PROGRAM PMPS_Arbiter
VAR
	
	fbPhotonEnergyWatcher	:	FB_PhotonEnergyWatcher;
	
	fbMPSInterface	:	FB_BeamClassOutputs;
    
    fbCuInterface	:	FB_CTLS_Outputs;
	
	(* Subsystem requests use this FB and a pragma link to pass their requests to the arbiter.
	The fb is called on each cycle and updates the arbiter with the current BP set requested 
	from the subsystem PLC.*)
	//<TODO> make this so it does input and output to the IF
	{attribute 'TcLinkTo' := '.i_RequestedBP:=TIIB[SubSysPLC1]^IO Inputs^RequestedBP; 
                                .o_CurrentBP:=TIIB[SubSysPLC1]^IO Outputs^CurrentBP;
                                .i_Connected:=TIIB[SubSysPLC1]^SYNC Inputs^External device not connected;
                                .i_WcState:=TIIB[SubSysPLC1]^WcState^WcState;
                                .i_TxPDOState:=TIIB[SubSysPLC1]^SYNC Inputs^TxPDO state;
                                '}
	fbSubSys1_PMPS_IO : FB_ArbiterToSubSys_IO := (RequestingSystemID := 16#FF0F);
	
	{attribute 'TcLinkTo' := '.i_RequestedBP:=TIIB[SubSysPLC2]^IO Inputs^RequestedBP;
                                .i_xNewRequest:=TIIB[SubSysPLC2]^IO Inputs^xNewRequest; 
                                .o_CurrentBP:=TIIB[SubSysPLC2]^IO Outputs^CurrentBP;
                                .i_Connected:=TIIB[SubSysPLC2]^SYNC Inputs^External device not connected;
                                .i_WcState:=TIIB[SubSysPLC2]^WcState^WcState;
                                .i_TxPDOState:=TIIB[SubSysPLC2]^SYNC Inputs^TxPDO state;
                                .i_TxPDOToggle:=TIIB[SubSysPLC2]^SYNC Inputs^TxPDO toggle;
                                '}
	fbSubSys2_PMPS_IO : FB_ArbiterToSubSys_IO := (RequestingSystemID := 16#FF10);
    
    fbBPRequestor : FB_BPRequestor;
	
	AttemptReset : TON := (PT:=T#1s);
    
    anothervar : bool;
    testFF : FB_FastFault;
    
    logging_active : BOOL;
    cycle : INT;
    
    {attribute 'pytmc' := '
		pv: @(PREFIX):PhotonEnergy
        link: ~
	'}
    fPhotonEnergy : REAL;
    
    {attribute 'pytmc' := '
		pv: @(PREFIX):PhotonEnergySeverity
        link: ~.SEVR
	'}
    iPhotonEnergySeverity : INT;
	
END_VAR


// Updating arbiter with subsystem requests.
fbSubSys1_PMPS_IO(Arbiter:=GVL.g_fbArbiter1, fbFFHWO:=GVL.g_FastFaultOutput1, Reset:=GVL.AttemptReset);

fbSubSys2_PMPS_IO(Arbiter:=GVL.g_fbArbiter1, fbFFHWO:=GVL.g_FastFaultOutput1, Reset:=GVL.AttemptReset);

// Example with attenuator peel-off
//////////////////////////////////

// Beam parameter requestor
fbBPRequestor(Arbiter:=GVL.g_fbArbiter1);

// Request beam class
fbMPSInterface(nBeamClass := 5);

// Request Cu beam rate
fbCuInterface(i_ArbiterBP := ReqBP);


// Keep an eye on the photon energy
fbPhotonEnergyWatcher(i_stCurrentBeamParams	:= PMPS_GVL.stCurrentBeamParameters,
					i_stRequestedBeamParams := ReqBP,
					io_fbFFHWO:= GVL.g_FastFaultOutput1,
                    i_xReset := GVL.AttemptReset);

AttemptReset(IN:=fbPhotonEnergyWatcher.xPhotonEnergyWithinBounds, Q=>GVL.AttemptReset);

// Trip a fast fault periodically
testFF(io_fbFFHWO:= g_FastFaultOutput1);
testFF.i_xOK := (cycle mod 1000) = 0;
cycle := cycle + 1;

g_FastFaultOutput1.EvaluateVetos();

IF logging_active THEN
    g_FastFaultOutput1.ExecuteLogging();
END_IF

END_PROGRAM

(* stored: Version 1.1.0.1, ProductVersion 3.1.4022.18
   POU PMPS_Arbiter: Id {91ae890b-11cc-4d41-83ec-edc5b802c784}, SpecialFunc None *)
